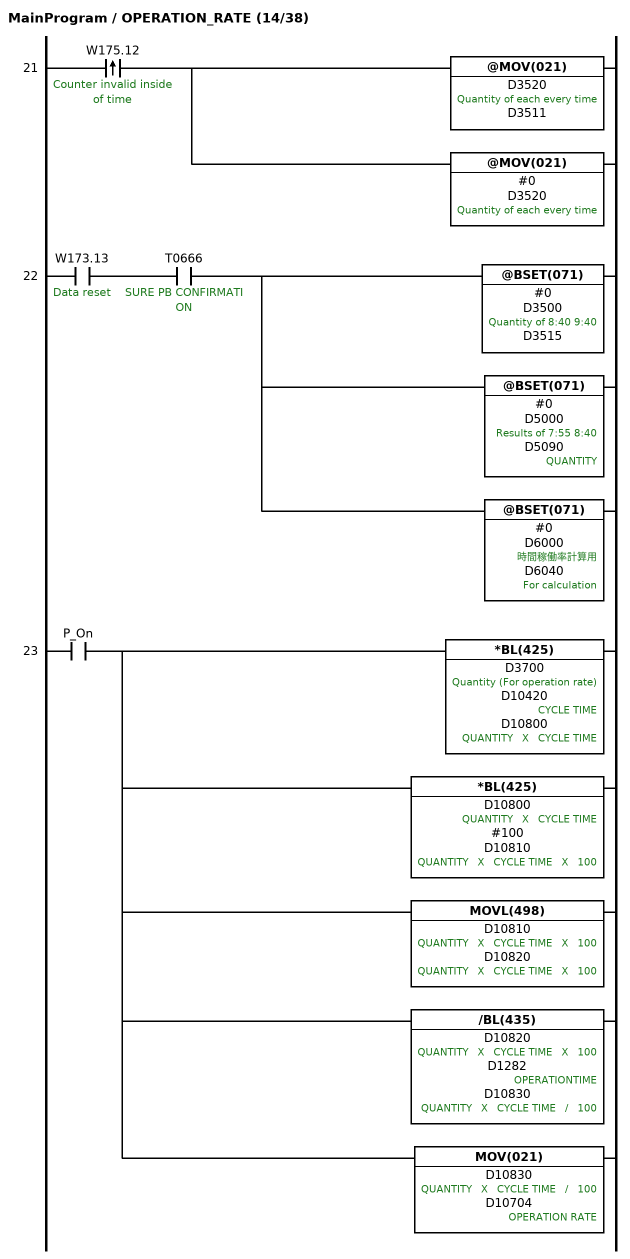
; [picture p264: MainProgram / OPERATION_RATE, rungs 21-23]
; rung 21
@LD W175.12  ; Counter invalid inside of time
@MOV(021) D3520 D3511  ; Quantity of each every time
@MOV(021) #0 D3520  ; Quantity of each every time
; rung 22
LD W173.13  ; Data reset
AND T0666  ; SURE PB CONFIRMATION
@BSET(071) #0 D3500 D3515  ; Quantity of 8:40 9:40
@BSET(071) #0 D5000 D5090  ; Results of 7:55 8:40, QUANTITY
@BSET(071) #0 D6000 D6040  ; 時間稼働率計算用, For calculation
; rung 23
LD P_On
*BL(425) D3700 D10420 D10800  ; Quantity (For operation rate), CYCLE TIME, QUANTITY   X   CYCLE TIME
*BL(425) D10800 #100 D10810  ; QUANTITY   X   CYCLE TIME, QUANTITY   X   CYCLE TIME   X   100
MOVL(498) D10810 D10820  ; QUANTITY   X   CYCLE TIME   X   100
/BL(435) D10820 D1282 D10830  ; QUANTITY   X   CYCLE TIME   X   100, OPERATIONTIME, QUANTITY   X   CYCLE TIME   /   100
MOV(021) D10830 D10704  ; QUANTITY   X   CYCLE TIME   /   100, OPERATION RATE

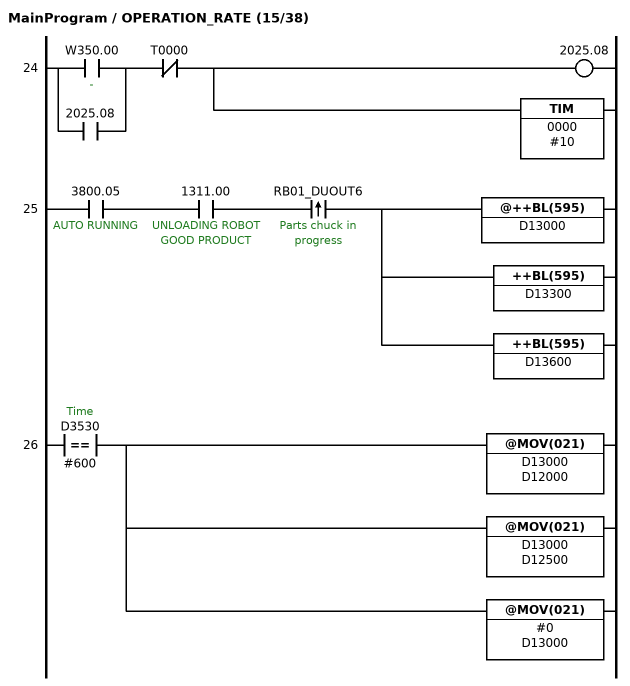
; rung 24
LD W350.00  ; -
OR 2025.08
ANDNOT T0000
OUT 2025.08
TIM 0000 #10
; rung 25
LD 3800.05  ; AUTO RUNNING
AND 1311.00  ; UNLOADING ROBOT GOOD PRODUCT
@AND RB01_DUOUT6  ; Parts chuck in progress
@++BL(595) D13000
++BL(595) D13300
++BL(595) D13600
; rung 26
LD=L(301) D3530 #600  ; Time
@MOV(021) D13000 D12000
@MOV(021) D13000 D12500
@MOV(021) #0 D13000

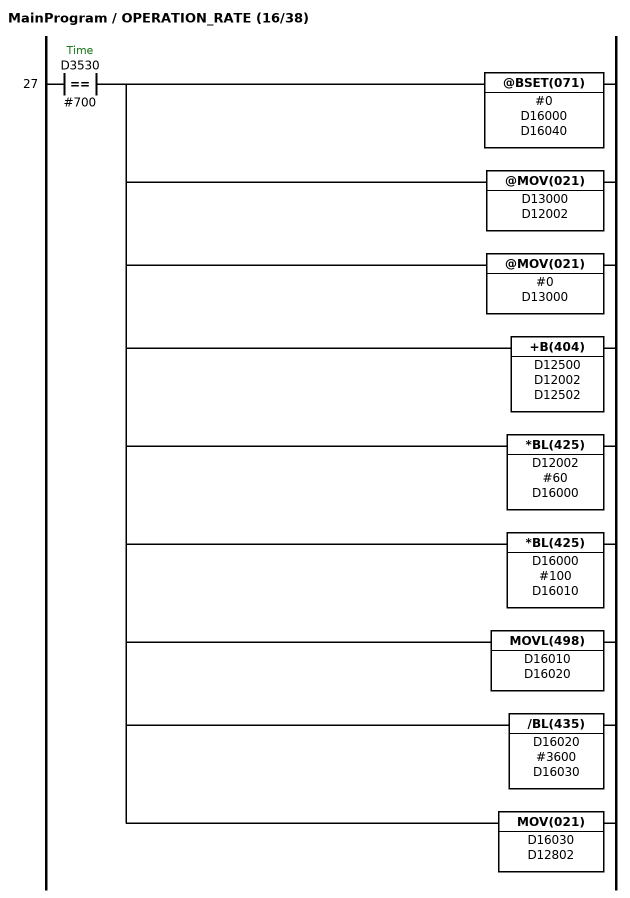
; rung 27
LD=L(301) D3530 #700  ; Time
@BSET(071) #0 D16000 D16040
@MOV(021) D13000 D12002
@MOV(021) #0 D13000
+B(404) D12500 D12002 D12502
*BL(425) D12002 #60 D16000
*BL(425) D16000 #100 D16010
MOVL(498) D16010 D16020
/BL(435) D16020 #3600 D16030
MOV(021) D16030 D12802

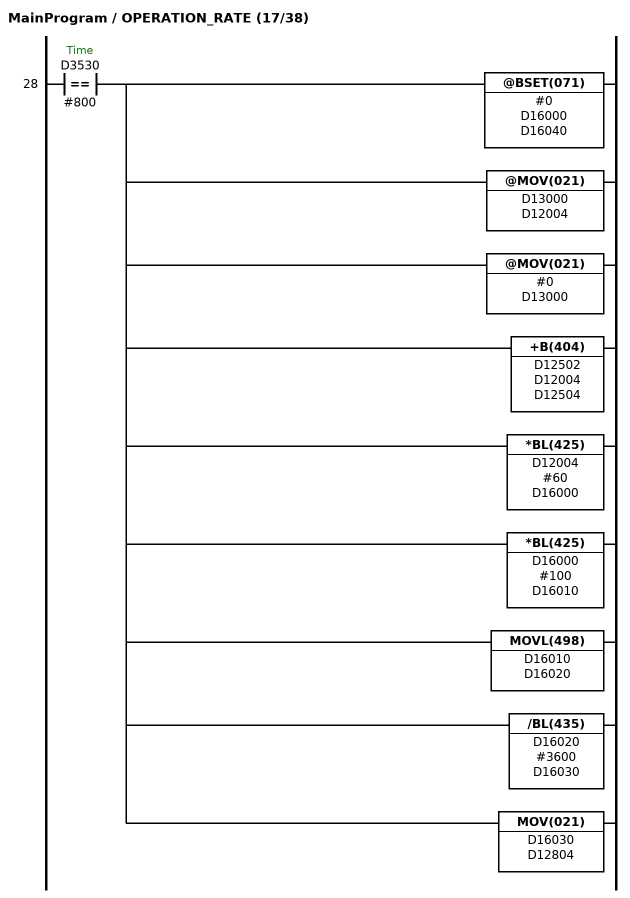
; rung 28
LD=L(301) D3530 #800  ; Time
@BSET(071) #0 D16000 D16040
@MOV(021) D13000 D12004
@MOV(021) #0 D13000
+B(404) D12502 D12004 D12504
*BL(425) D12004 #60 D16000
*BL(425) D16000 #100 D16010
MOVL(498) D16010 D16020
/BL(435) D16020 #3600 D16030
MOV(021) D16030 D12804

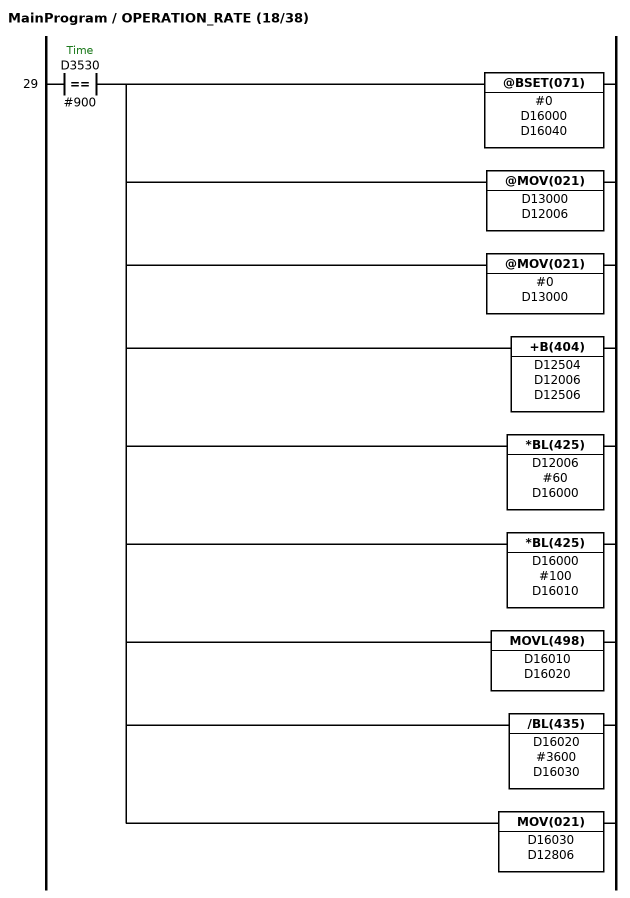
; rung 29
LD=L(301) D3530 #900  ; Time
@BSET(071) #0 D16000 D16040
@MOV(021) D13000 D12006
@MOV(021) #0 D13000
+B(404) D12504 D12006 D12506
*BL(425) D12006 #60 D16000
*BL(425) D16000 #100 D16010
MOVL(498) D16010 D16020
/BL(435) D16020 #3600 D16030
MOV(021) D16030 D12806

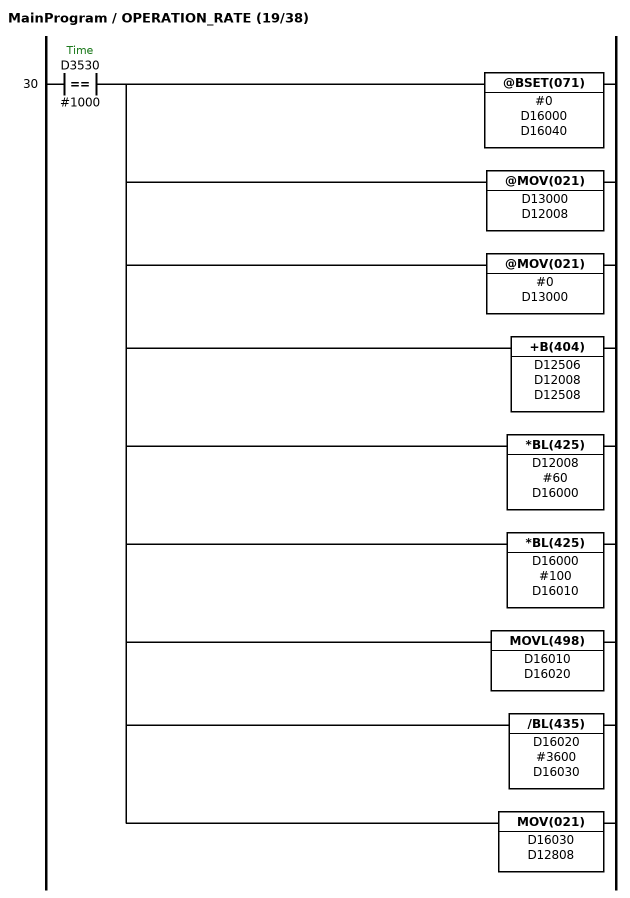
; rung 30
LD=L(301) D3530 #1000  ; Time
@BSET(071) #0 D16000 D16040
@MOV(021) D13000 D12008
@MOV(021) #0 D13000
+B(404) D12506 D12008 D12508
*BL(425) D12008 #60 D16000
*BL(425) D16000 #100 D16010
MOVL(498) D16010 D16020
/BL(435) D16020 #3600 D16030
MOV(021) D16030 D12808

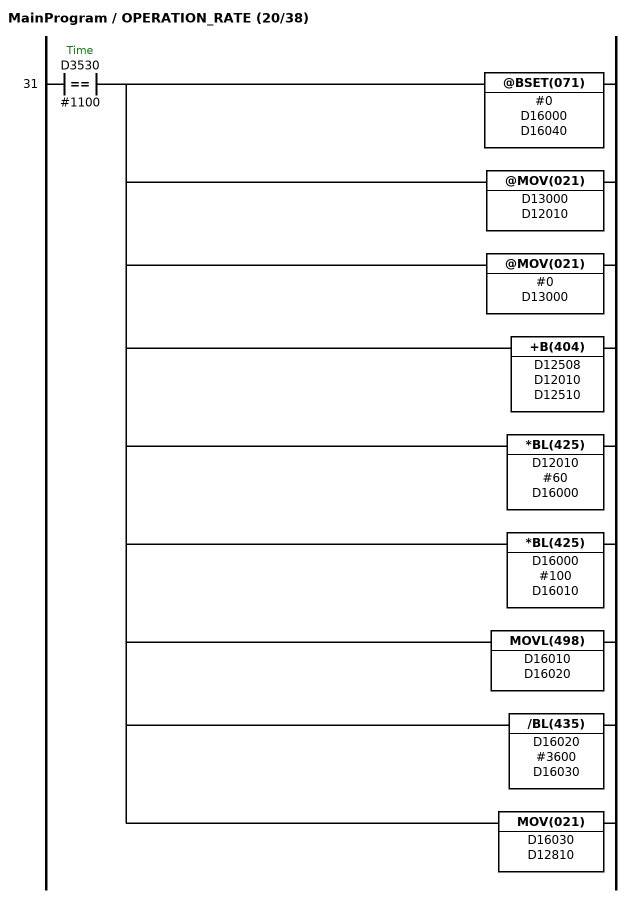
; rung 31
LD=L(301) D3530 #1100  ; Time
@BSET(071) #0 D16000 D16040
@MOV(021) D13000 D12010
@MOV(021) #0 D13000
+B(404) D12508 D12010 D12510
*BL(425) D12010 #60 D16000
*BL(425) D16000 #100 D16010
MOVL(498) D16010 D16020
/BL(435) D16020 #3600 D16030
MOV(021) D16030 D12810

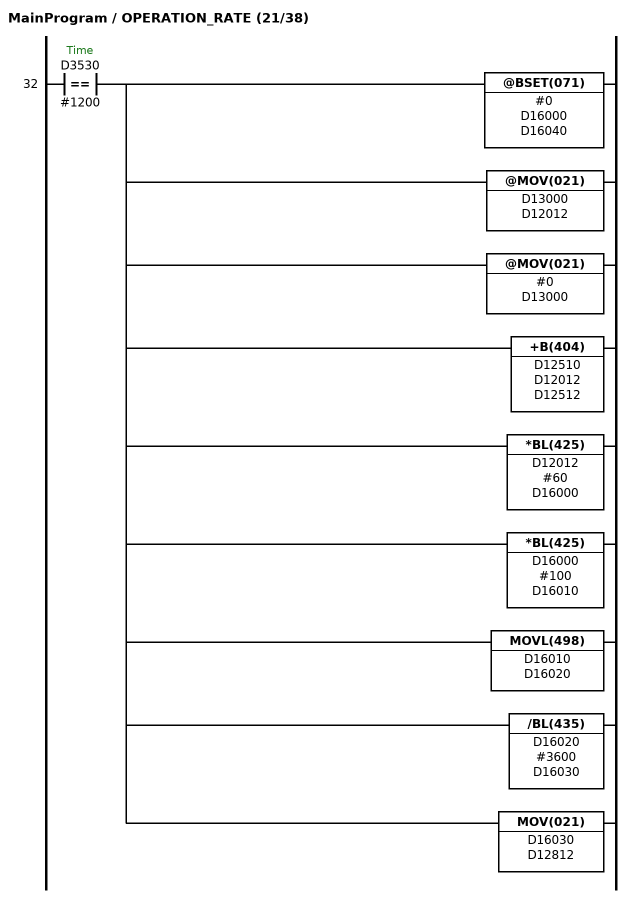
; rung 32
LD=L(301) D3530 #1200  ; Time
@BSET(071) #0 D16000 D16040
@MOV(021) D13000 D12012
@MOV(021) #0 D13000
+B(404) D12510 D12012 D12512
*BL(425) D12012 #60 D16000
*BL(425) D16000 #100 D16010
MOVL(498) D16010 D16020
/BL(435) D16020 #3600 D16030
MOV(021) D16030 D12812

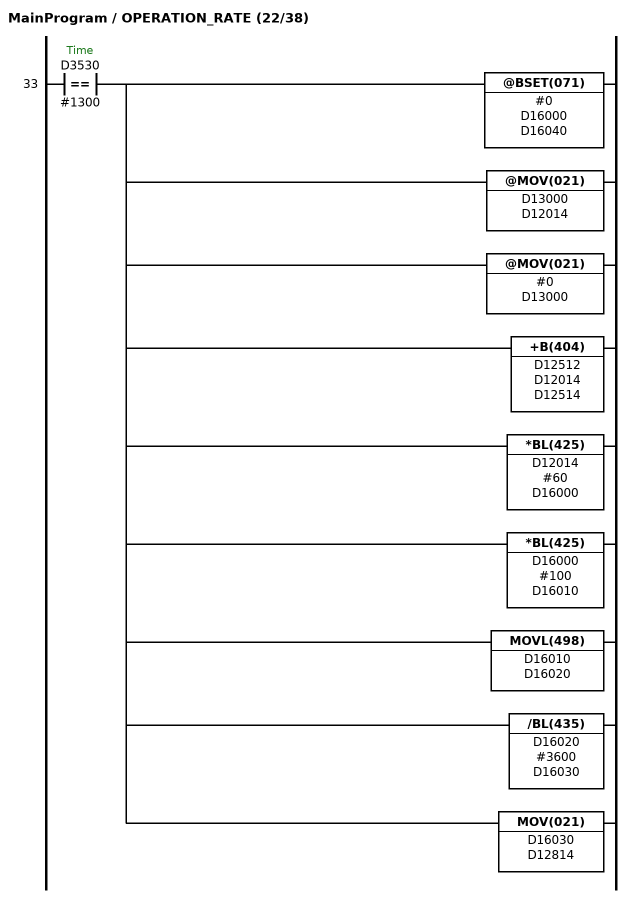
; rung 33
LD=L(301) D3530 #1300  ; Time
@BSET(071) #0 D16000 D16040
@MOV(021) D13000 D12014
@MOV(021) #0 D13000
+B(404) D12512 D12014 D12514
*BL(425) D12014 #60 D16000
*BL(425) D16000 #100 D16010
MOVL(498) D16010 D16020
/BL(435) D16020 #3600 D16030
MOV(021) D16030 D12814

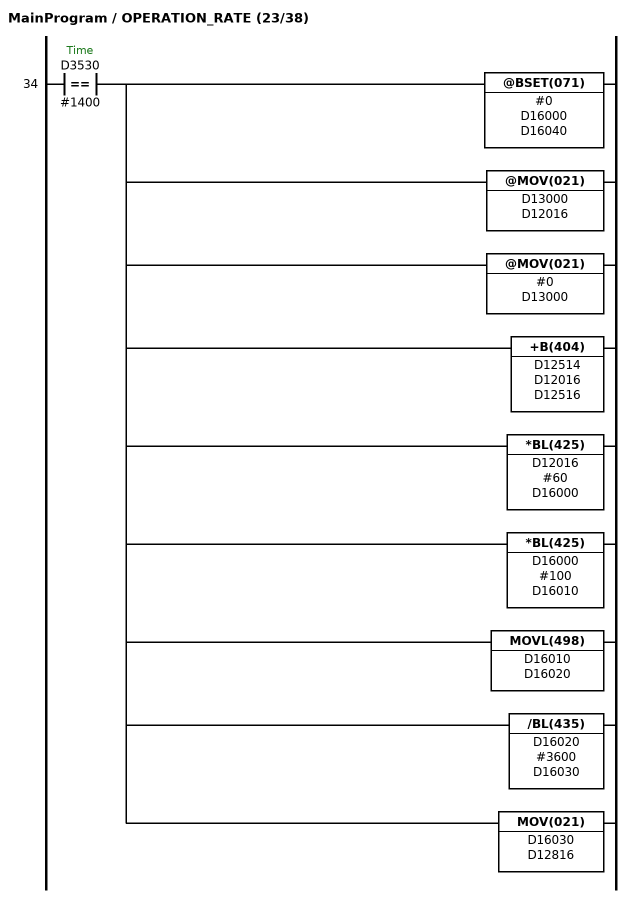
; rung 34
LD=L(301) D3530 #1400  ; Time
@BSET(071) #0 D16000 D16040
@MOV(021) D13000 D12016
@MOV(021) #0 D13000
+B(404) D12514 D12016 D12516
*BL(425) D12016 #60 D16000
*BL(425) D16000 #100 D16010
MOVL(498) D16010 D16020
/BL(435) D16020 #3600 D16030
MOV(021) D16030 D12816

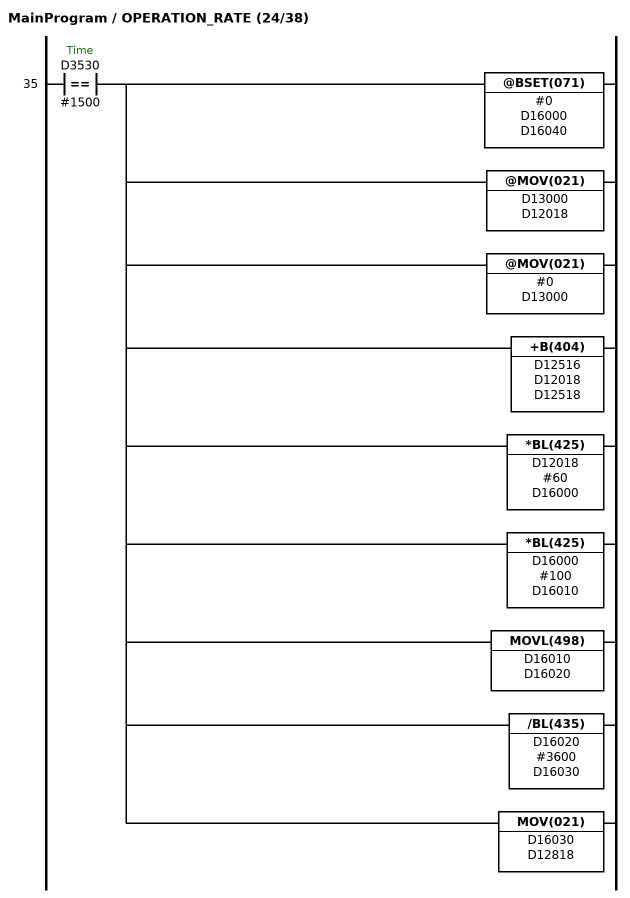
; rung 35
LD=L(301) D3530 #1500  ; Time
@BSET(071) #0 D16000 D16040
@MOV(021) D13000 D12018
@MOV(021) #0 D13000
+B(404) D12516 D12018 D12518
*BL(425) D12018 #60 D16000
*BL(425) D16000 #100 D16010
MOVL(498) D16010 D16020
/BL(435) D16020 #3600 D16030
MOV(021) D16030 D12818

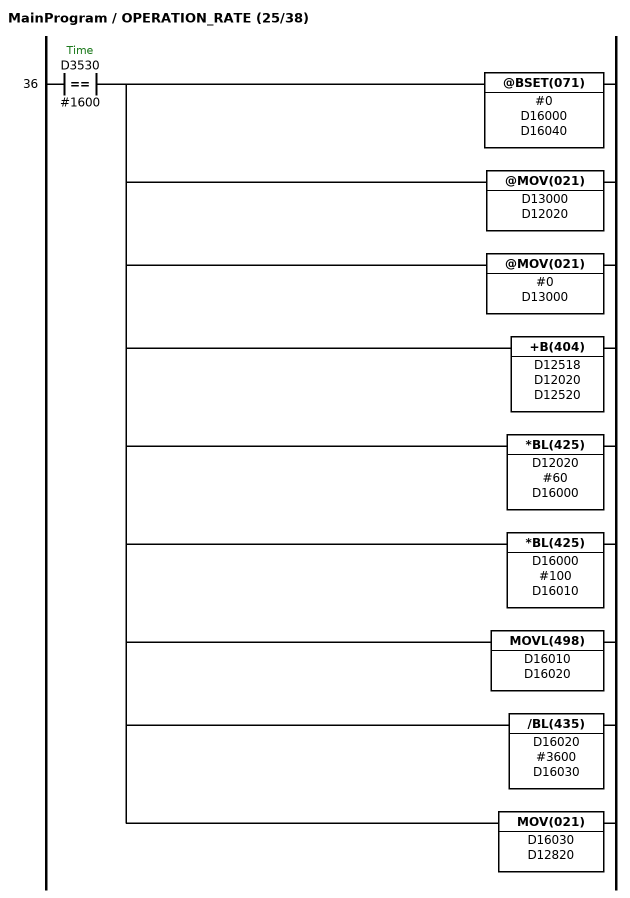
; rung 36
LD=L(301) D3530 #1600  ; Time
@BSET(071) #0 D16000 D16040
@MOV(021) D13000 D12020
@MOV(021) #0 D13000
+B(404) D12518 D12020 D12520
*BL(425) D12020 #60 D16000
*BL(425) D16000 #100 D16010
MOVL(498) D16010 D16020
/BL(435) D16020 #3600 D16030
MOV(021) D16030 D12820

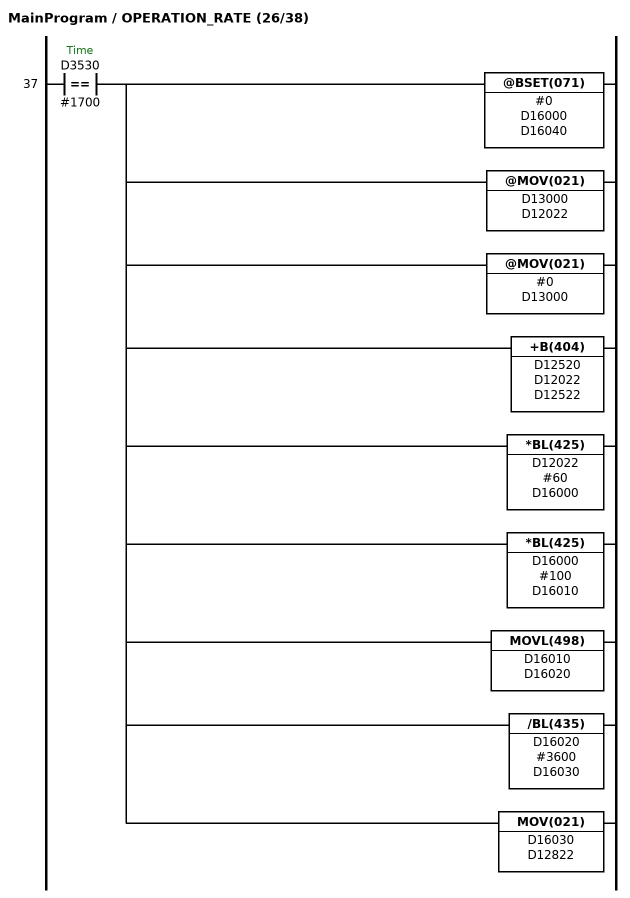
; rung 37
LD=L(301) D3530 #1700  ; Time
@BSET(071) #0 D16000 D16040
@MOV(021) D13000 D12022
@MOV(021) #0 D13000
+B(404) D12520 D12022 D12522
*BL(425) D12022 #60 D16000
*BL(425) D16000 #100 D16010
MOVL(498) D16010 D16020
/BL(435) D16020 #3600 D16030
MOV(021) D16030 D12822

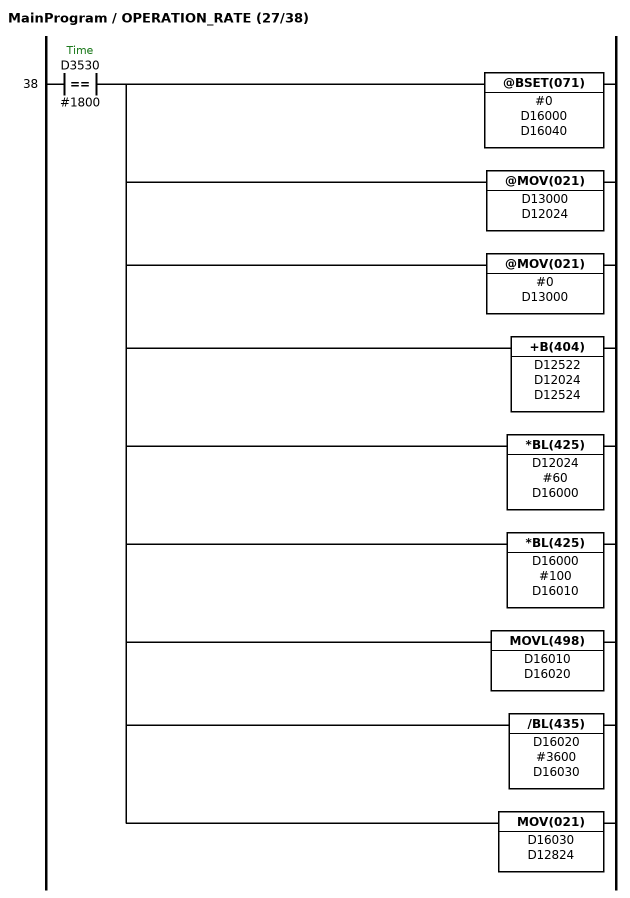
; rung 38
LD=L(301) D3530 #1800  ; Time
@BSET(071) #0 D16000 D16040
@MOV(021) D13000 D12024
@MOV(021) #0 D13000
+B(404) D12522 D12024 D12524
*BL(425) D12024 #60 D16000
*BL(425) D16000 #100 D16010
MOVL(498) D16010 D16020
/BL(435) D16020 #3600 D16030
MOV(021) D16030 D12824

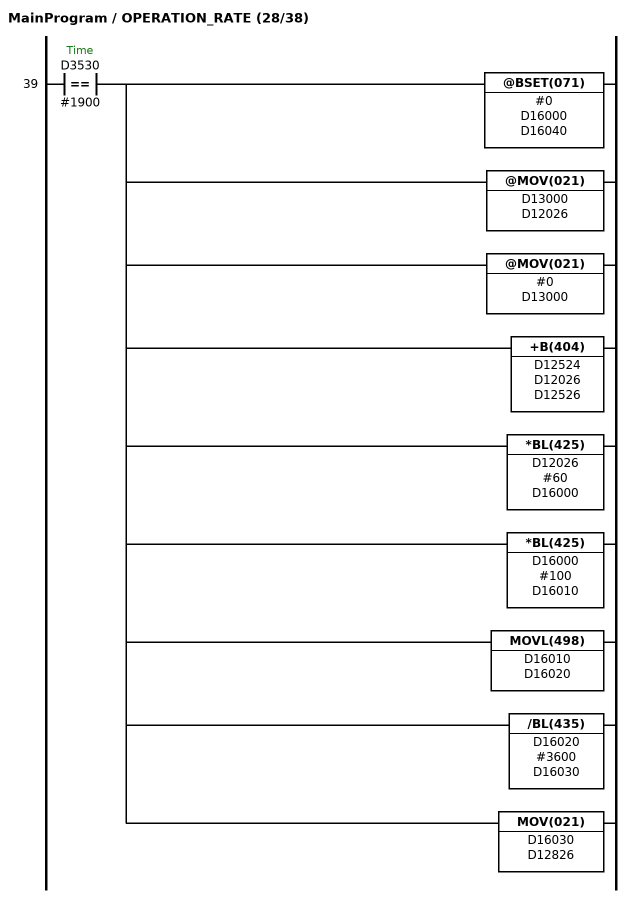
; rung 39
LD=L(301) D3530 #1900  ; Time
@BSET(071) #0 D16000 D16040
@MOV(021) D13000 D12026
@MOV(021) #0 D13000
+B(404) D12524 D12026 D12526
*BL(425) D12026 #60 D16000
*BL(425) D16000 #100 D16010
MOVL(498) D16010 D16020
/BL(435) D16020 #3600 D16030
MOV(021) D16030 D12826

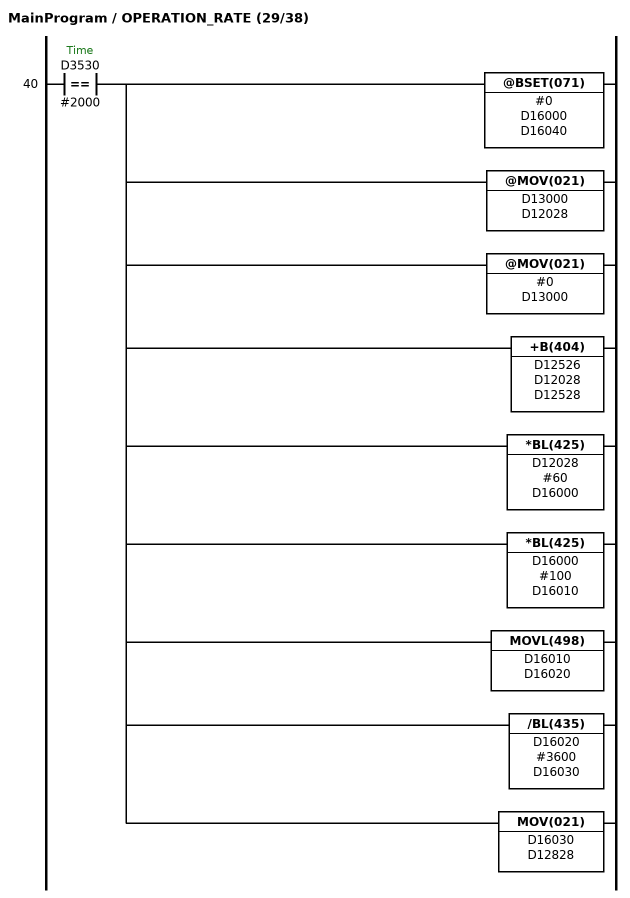
; rung 40
LD=L(301) D3530 #2000  ; Time
@BSET(071) #0 D16000 D16040
@MOV(021) D13000 D12028
@MOV(021) #0 D13000
+B(404) D12526 D12028 D12528
*BL(425) D12028 #60 D16000
*BL(425) D16000 #100 D16010
MOVL(498) D16010 D16020
/BL(435) D16020 #3600 D16030
MOV(021) D16030 D12828

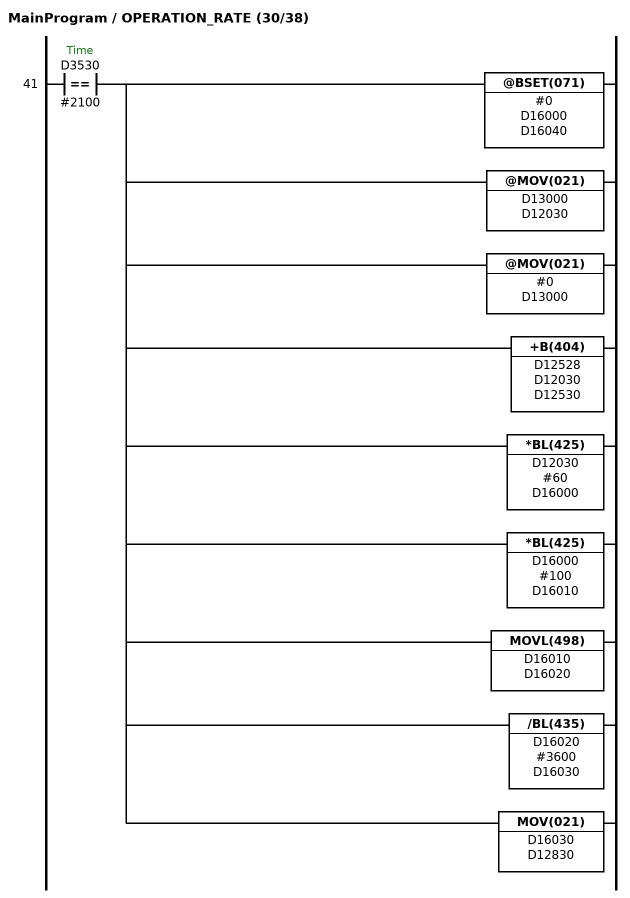
; rung 41
LD=L(301) D3530 #2100  ; Time
@BSET(071) #0 D16000 D16040
@MOV(021) D13000 D12030
@MOV(021) #0 D13000
+B(404) D12528 D12030 D12530
*BL(425) D12030 #60 D16000
*BL(425) D16000 #100 D16010
MOVL(498) D16010 D16020
/BL(435) D16020 #3600 D16030
MOV(021) D16030 D12830

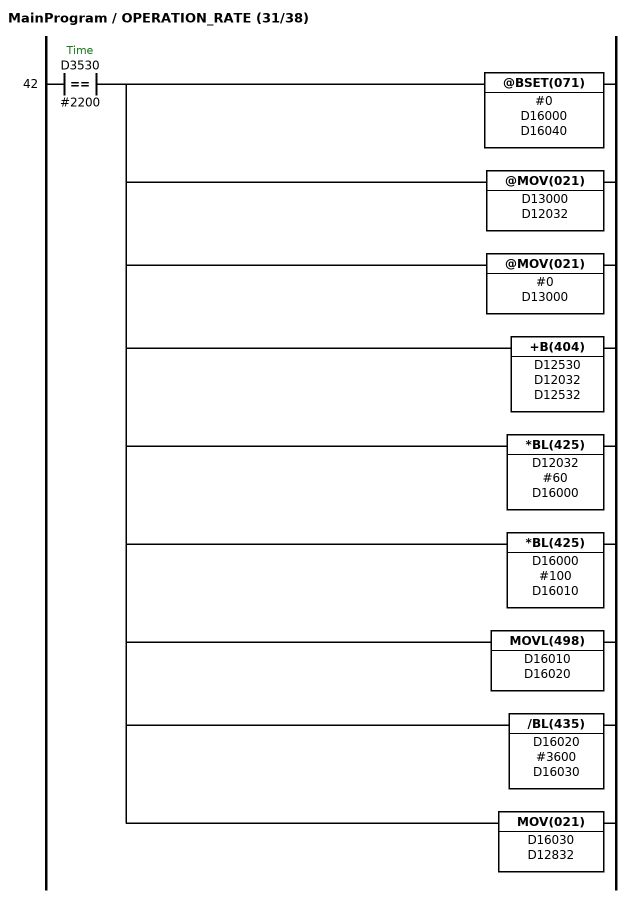
; rung 42
LD=L(301) D3530 #2200  ; Time
@BSET(071) #0 D16000 D16040
@MOV(021) D13000 D12032
@MOV(021) #0 D13000
+B(404) D12530 D12032 D12532
*BL(425) D12032 #60 D16000
*BL(425) D16000 #100 D16010
MOVL(498) D16010 D16020
/BL(435) D16020 #3600 D16030
MOV(021) D16030 D12832

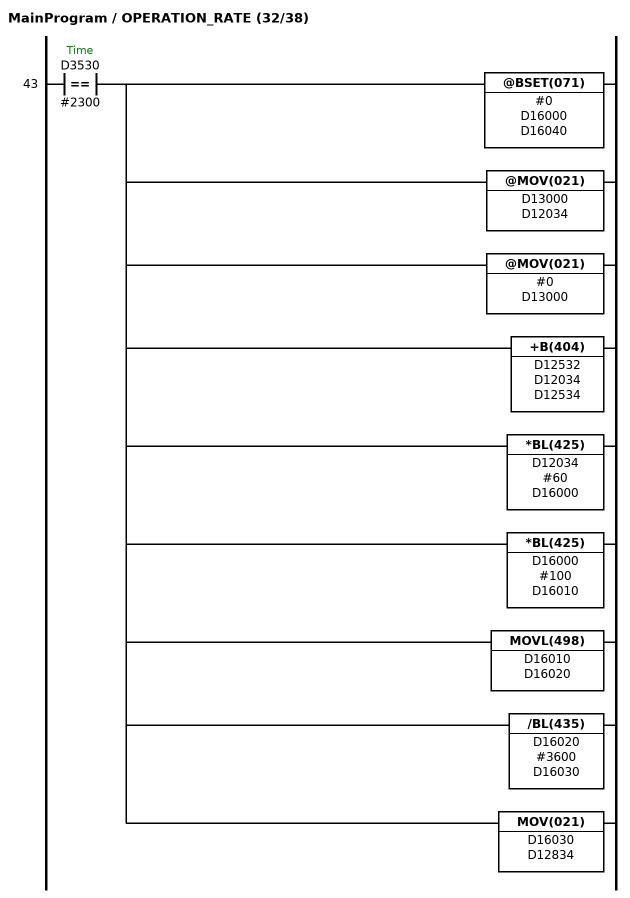
; rung 43
LD=L(301) D3530 #2300  ; Time
@BSET(071) #0 D16000 D16040
@MOV(021) D13000 D12034
@MOV(021) #0 D13000
+B(404) D12532 D12034 D12534
*BL(425) D12034 #60 D16000
*BL(425) D16000 #100 D16010
MOVL(498) D16010 D16020
/BL(435) D16020 #3600 D16030
MOV(021) D16030 D12834

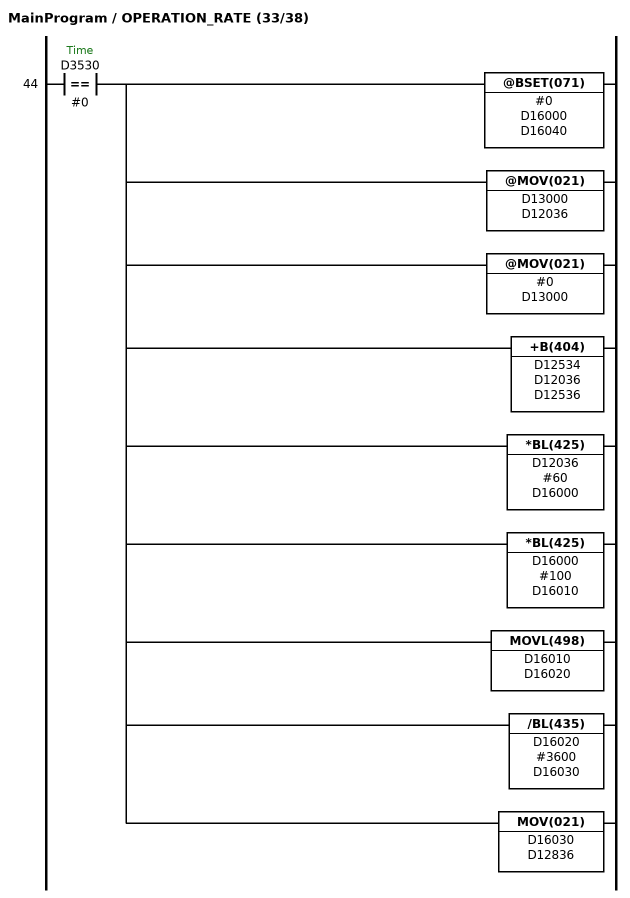
; rung 44
LD=L(301) D3530 #0  ; Time
@BSET(071) #0 D16000 D16040
@MOV(021) D13000 D12036
@MOV(021) #0 D13000
+B(404) D12534 D12036 D12536
*BL(425) D12036 #60 D16000
*BL(425) D16000 #100 D16010
MOVL(498) D16010 D16020
/BL(435) D16020 #3600 D16030
MOV(021) D16030 D12836

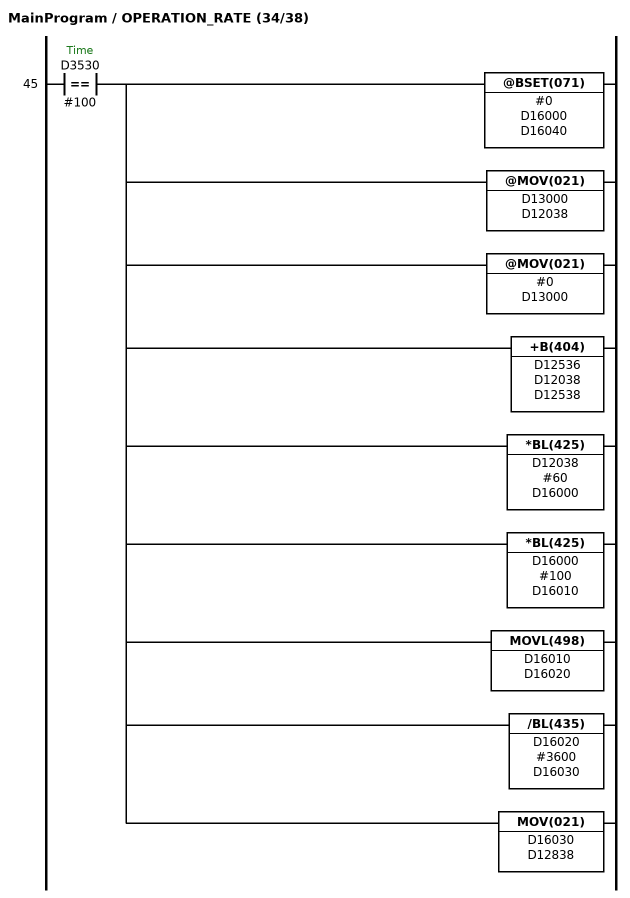
; rung 45
LD=L(301) D3530 #100  ; Time
@BSET(071) #0 D16000 D16040
@MOV(021) D13000 D12038
@MOV(021) #0 D13000
+B(404) D12536 D12038 D12538
*BL(425) D12038 #60 D16000
*BL(425) D16000 #100 D16010
MOVL(498) D16010 D16020
/BL(435) D16020 #3600 D16030
MOV(021) D16030 D12838

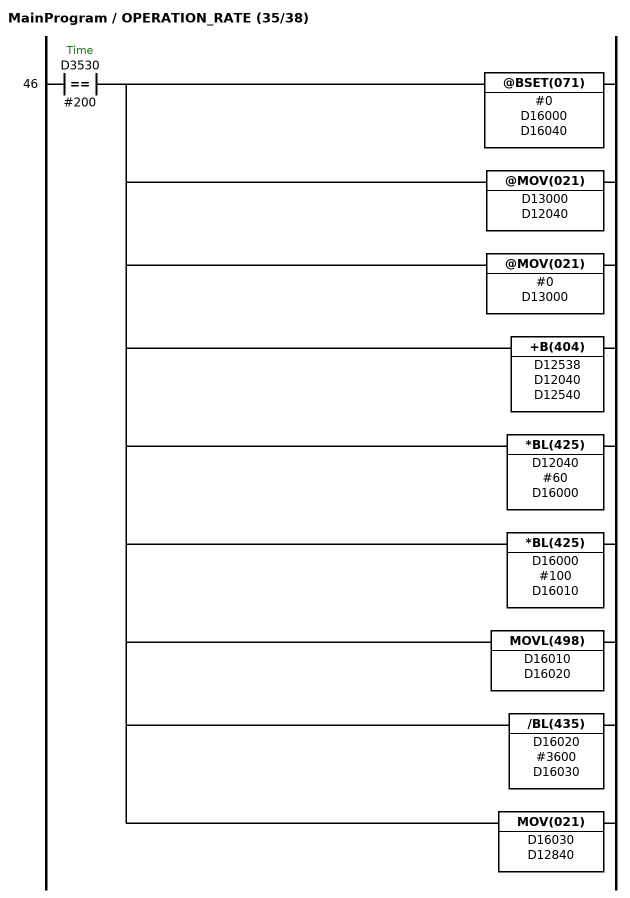
; rung 46
LD=L(301) D3530 #200  ; Time
@BSET(071) #0 D16000 D16040
@MOV(021) D13000 D12040
@MOV(021) #0 D13000
+B(404) D12538 D12040 D12540
*BL(425) D12040 #60 D16000
*BL(425) D16000 #100 D16010
MOVL(498) D16010 D16020
/BL(435) D16020 #3600 D16030
MOV(021) D16030 D12840

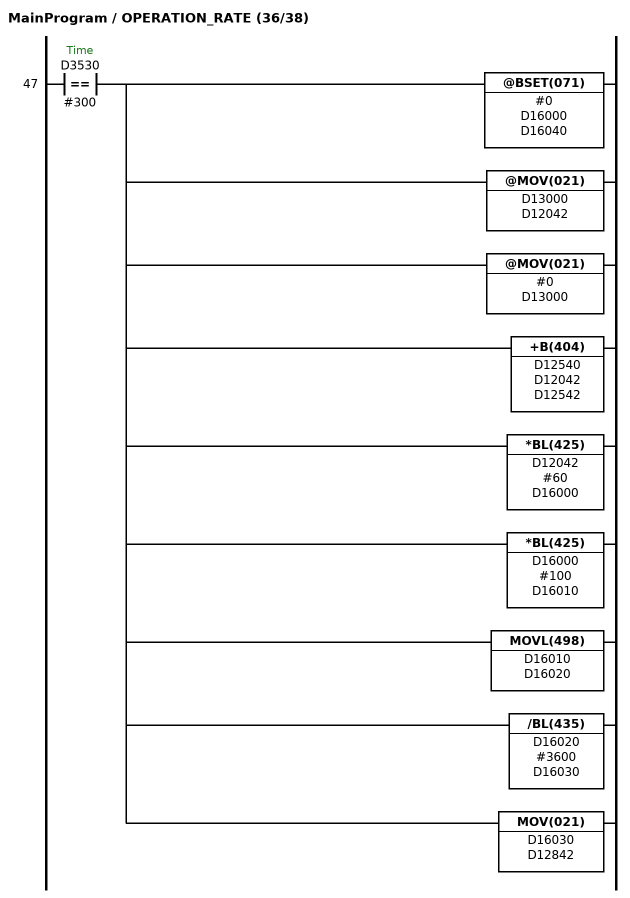
; rung 47
LD=L(301) D3530 #300  ; Time
@BSET(071) #0 D16000 D16040
@MOV(021) D13000 D12042
@MOV(021) #0 D13000
+B(404) D12540 D12042 D12542
*BL(425) D12042 #60 D16000
*BL(425) D16000 #100 D16010
MOVL(498) D16010 D16020
/BL(435) D16020 #3600 D16030
MOV(021) D16030 D12842

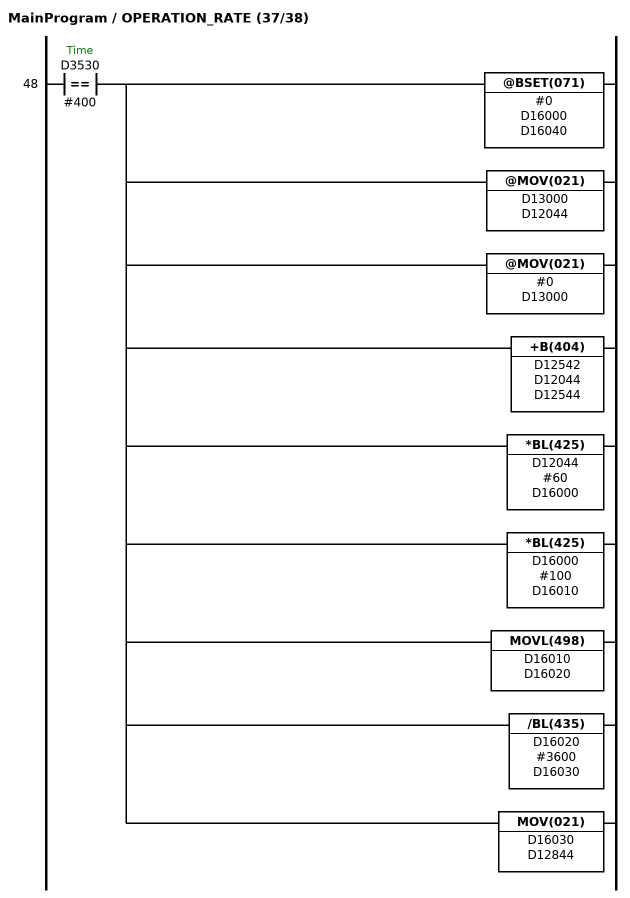
; rung 48
LD=L(301) D3530 #400  ; Time
@BSET(071) #0 D16000 D16040
@MOV(021) D13000 D12044
@MOV(021) #0 D13000
+B(404) D12542 D12044 D12544
*BL(425) D12044 #60 D16000
*BL(425) D16000 #100 D16010
MOVL(498) D16010 D16020
/BL(435) D16020 #3600 D16030
MOV(021) D16030 D12844

